TEXTLIST AxesMoveUnitsTextList
  0 = 'degrees'
  1 = 'rad'
  2 = 'arcsec'
   = ''
END_TEXTLIST

(* stored: Version 1.1.0.1, ProductVersion 3.1.4019.2
   TextList AxesMoveUnitsTextList: Id {9c7b5ab0-7add-41ff-8650-01dbd7878aae} *)
